IF in < DatatypeLimits.MIN_VALUE_OF_LREAL_WHICH_CAN_BE_HELD_IN_A_UDINT THEN
	RETURN;
END_IF

out := LREAL_TO_UDINT(in);
TryConvert_LREAL_TO_UDINT := TRUE;

END_FUNCTION

// ---- Converters/LREAL_TO_/TryConvert_LREAL_TO_ULINT.TcPOU
FUNCTION TryConvert_LREAL_TO_ULINT : BOOL
VAR_INPUT
	in : LREAL;
	out : REFERENCE TO ULINT;
END_VAR

IF in > DatatypeLimits.MAX_VALUE_OF_LREAL_WHICH_CAN_BE_HELD_IN_A_ULINT THEN
	RETURN;
END_IF

IF in < DatatypeLimits.MIN_VALUE_OF_LREAL_WHICH_CAN_BE_HELD_IN_A_ULINT THEN
	RETURN;
END_IF

out := LREAL_TO_ULINT(in);
TryConvert_LREAL_TO_ULINT := TRUE;

END_FUNCTION

// ---- Converters/LREAL_TO_/TryConvert_LREAL_TO_REAL.TcPOU
FUNCTION TryConvert_LREAL_TO_REAL : BOOL
VAR_INPUT
	in : LREAL;
	out : REFERENCE TO REAL;
END_VAR

IF in > DatatypeLimits.MAX_VALUE_OF_LREAL_WHICH_CAN_BE_HELD_IN_A_REAL THEN
	RETURN;
END_IF

IF in < DatatypeLimits.MIN_VALUE_OF_LREAL_WHICH_CAN_BE_HELD_IN_A_REAL THEN
	RETURN;
END_IF

out := LREAL_TO_REAL(in);
TryConvert_LREAL_TO_REAL := TRUE;

END_FUNCTION

// ---- Converters/LREAL_TO_/TryConvert_LREAL_TO_LREAL.TcPOU
FUNCTION TryConvert_LREAL_TO_LREAL : BOOL
VAR_INPUT
	in : LREAL;
	out : REFERENCE TO LREAL;
END_VAR

out := in;
TryConvert_LREAL_TO_LREAL := TRUE;

END_FUNCTION

// ---- Converters/LREAL_TO_/TryConvert_LREAL_TO_TIME.TcPOU
FUNCTION TryConvert_LREAL_TO_TIME : BOOL
VAR_INPUT
	in : LREAL;
	out : REFERENCE TO TIME;
END_VAR

IF in > DatatypeLimits.MAX_VALUE_OF_LREAL_WHICH_CAN_BE_HELD_IN_A_TIME THEN
	RETURN;
END_IF

IF in < DatatypeLimits.MIN_VALUE_OF_LREAL_WHICH_CAN_BE_HELD_IN_A_TIME THEN
	RETURN;
END_IF

out := LREAL_TO_TIME(in);
TryConvert_LREAL_TO_TIME := TRUE;

END_FUNCTION

// ---- Converters/LREAL_TO_/TryConvert_LREAL_TO_TOD.TcPOU
FUNCTION TryConvert_LREAL_TO_TOD : BOOL
VAR_INPUT
	in : LREAL;
	out : REFERENCE TO TOD;
END_VAR

IF in > DatatypeLimits.MAX_VALUE_OF_LREAL_WHICH_CAN_BE_HELD_IN_A_TOD THEN
	RETURN;
END_IF

IF in < DatatypeLimits.MIN_VALUE_OF_LREAL_WHICH_CAN_BE_HELD_IN_A_TOD THEN
	RETURN;
END_IF

out := LREAL_TO_TOD(in);
TryConvert_LREAL_TO_TOD := TRUE;

END_FUNCTION

// ---- Converters/LREAL_TO_/TryConvert_LREAL_TO_DT.TcPOU
FUNCTION TryConvert_LREAL_TO_DT : BOOL
VAR_INPUT
	in : LREAL;
	out : REFERENCE TO DT;
END_VAR

IF in > DatatypeLimits.MAX_VALUE_OF_LREAL_WHICH_CAN_BE_HELD_IN_A_DT THEN
	RETURN;
END_IF

IF in < DatatypeLimits.MIN_VALUE_OF_LREAL_WHICH_CAN_BE_HELD_IN_A_DT THEN
	RETURN;
END_IF

out := LREAL_TO_DT(in);
TryConvert_LREAL_TO_DT := TRUE;

END_FUNCTION

// ---- Converters/LREAL_TO_/TryConvert_LREAL_TO_STRING.TcPOU
FUNCTION TryConvert_LREAL_TO_STRING : BOOL
VAR_INPUT
	in : LREAL;
	out : REFERENCE TO STRING;
END_VAR

IF in > DatatypeLimits.MAX_VALUE_OF_LREAL_WHICH_CAN_BE_HELD_IN_A_STRING THEN
	RETURN;
END_IF

IF in < DatatypeLimits.MIN_VALUE_OF_LREAL_WHICH_CAN_BE_HELD_IN_A_STRING THEN
	RETURN;
END_IF

out := LREAL_TO_STRING(in);
TryConvert_LREAL_TO_STRING := TRUE;

END_FUNCTION

// ---- Converters/LWORD_TO_/TryConvert_LWORD_TO_BOOL.TcPOU
FUNCTION TryConvert_LWORD_TO_BOOL : BOOL
VAR_INPUT
	in : LWORD;
	out : REFERENCE TO BOOL;
END_VAR

out := LWORD_TO_BOOL(in);
TryConvert_LWORD_TO_BOOL := TRUE;

END_FUNCTION

// ---- Converters/LWORD_TO_/TryConvert_LWORD_TO_BYTE.TcPOU
FUNCTION TryConvert_LWORD_TO_BYTE : BOOL
VAR_INPUT
	in : LWORD;
	out : REFERENCE TO BYTE;
END_VAR

IF in > DatatypeLimits.MAX_VALUE_OF_LWORD_WHICH_CAN_BE_HELD_IN_A_BYTE THEN
	RETURN;
END_IF

out := LWORD_TO_BYTE(in);
TryConvert_LWORD_TO_BYTE := TRUE;

END_FUNCTION

// ---- Converters/LWORD_TO_/TryConvert_LWORD_TO_DATE.TcPOU
FUNCTION TryConvert_LWORD_TO_DATE : BOOL
VAR_INPUT
	in : LWORD;
	out : REFERENCE TO DATE;
END_VAR

IF in > DatatypeLimits.MAX_VALUE_OF_LWORD_WHICH_CAN_BE_HELD_IN_A_DATE THEN
	RETURN;
END_IF

out := LWORD_TO_DATE(in);
TryConvert_LWORD_TO_DATE := TRUE;

END_FUNCTION

// ---- Converters/LWORD_TO_/TryConvert_LWORD_TO_Destination.TcPOU
FUNCTION TryConvert_LWORD_TO_Destination : BOOL
VAR_INPUT
	in : LWORD;
	out : ANY;
END_VAR
VAR
	convertResult : BOOL := FALSE;
	convertAddress : PVOID;
	_BOOL : BOOL;
	_BYTE : BYTE;
	_WORD : WORD;
	_DWORD : DWORD;
	_LWORD : LWORD;
	_SINT : SINT;
	_INT : INT;
	_DINT : DINT;
	_LINT : LINT;
	_USINT : USINT;
	_UINT : UINT;
	_UDINT : UDINT;
	_ULINT : ULINT;
	_REAL : REAL;
	_LREAL : LREAL;
	_TIME : TIME;
	_TOD : TOD;
	_DATE : DATE;
	_DT : DT;
	_STRING : STRING;
END_VAR

CASE out.TypeClass OF
	__SYSTEM.TYPE_CLASS.TYPE_BOOL:
	
	convertResult := TryConvert_LWORD_TO_BOOL(in, _BOOL);
	IF convertResult THEN
		convertAddress := ADR(_BOOL);
	END_IF
	
	__SYSTEM.TYPE_CLASS.TYPE_BYTE:
	
	convertResult := TryConvert_LWORD_TO_BYTE(in, _BYTE);
	IF convertResult THEN
		convertAddress := ADR(_BYTE);
	END_IF
	
	__SYSTEM.TYPE_CLASS.TYPE_WORD:
	
	convertResult := TryConvert_LWORD_TO_WORD(in, _WORD);
	IF convertResult THEN
		convertAddress := ADR(_WORD);
	END_IF
	
	__SYSTEM.TYPE_CLASS.TYPE_DWORD:
	
	convertResult := TryConvert_LWORD_TO_DWORD(in, _DWORD);
	IF convertResult THEN
		convertAddress := ADR(_DWORD);
	END_IF
	
	__SYSTEM.TYPE_CLASS.TYPE_LWORD:
	
	convertResult := TryConvert_LWORD_TO_LWORD(in, _LWORD);
	IF convertResult THEN
		convertAddress := ADR(_LWORD);
	END_IF
	
	__SYSTEM.TYPE_CLASS.TYPE_SINT:
	
	convertResult := TryConvert_LWORD_TO_SINT(in, _SINT);
	IF convertResult THEN
		convertAddress := ADR(_SINT);
	END_IF
	
	__SYSTEM.TYPE_CLASS.TYPE_INT:
	
	convertResult := TryConvert_LWORD_TO_INT(in, _INT);
	IF convertResult THEN
		convertAddress := ADR(_INT);
	END_IF
	
	__SYSTEM.TYPE_CLASS.TYPE_DINT:
	
	convertResult := TryConvert_LWORD_TO_DINT(in, _DINT);
	IF convertResult THEN
		convertAddress := ADR(_DINT);
	END_IF
	
	__SYSTEM.TYPE_CLASS.TYPE_LINT:
	
	convertResult := TryConvert_LWORD_TO_LINT(in, _LINT);
	IF convertResult THEN
		convertAddress := ADR(_LINT);
	END_IF
	
	__SYSTEM.TYPE_CLASS.TYPE_USINT:
	
	convertResult := TryConvert_LWORD_TO_USINT(in, _USINT);
	IF convertResult THEN
		convertAddress := ADR(_USINT);
	END_IF
	
	__SYSTEM.TYPE_CLASS.TYPE_UINT:
	
	convertResult := TryConvert_LWORD_TO_UINT(in, _UINT);
	IF convertResult THEN
		convertAddress := ADR(_UINT);
	END_IF
	
	__SYSTEM.TYPE_CLASS.TYPE_UDINT:
	
	convertResult := TryConvert_LWORD_TO_UDINT(in, _UDINT);
	IF convertResult THEN
		convertAddress := ADR(_UDINT);
	END_IF
	
	__SYSTEM.TYPE_CLASS.TYPE_ULINT:
	
	convertResult := TryConvert_LWORD_TO_ULINT(in, _ULINT);
	IF convertResult THEN
		convertAddress := ADR(_ULINT);
	END_IF
	
	__SYSTEM.TYPE_CLASS.TYPE_REAL:
	
	convertResult := TryConvert_LWORD_TO_REAL(in, _REAL);
	IF convertResult THEN
		convertAddress := ADR(_REAL);
	END_IF
	
	__SYSTEM.TYPE_CLASS.TYPE_LREAL:
	
	convertResult := TryConvert_LWORD_TO_LREAL(in, _LREAL);
	IF convertResult THEN
		convertAddress := ADR(_LREAL);
	END_IF
	
	__SYSTEM.TYPE_CLASS.TYPE_TIME:
	
	convertResult := TryConvert_LWORD_TO_TIME(in, _TIME);
	IF convertResult THEN
		convertAddress := ADR(_TIME);
	END_IF
	
	__SYSTEM.TYPE_CLASS.TYPE_TIMEOFDAY:
	
	convertResult := TryConvert_LWORD_TO_TOD(in, _TOD);
	IF convertResult THEN
		convertAddress := ADR(_TOD);
	END_IF
	
	__SYSTEM.TYPE_CLASS.TYPE_DATE:
	
	convertResult := TryConvert_LWORD_TO_DATE(in, _DATE);
	IF convertResult THEN
		convertAddress := ADR(_DATE);
	END_IF
	
	__SYSTEM.TYPE_CLASS.TYPE_DATEANDTIME:
	
	convertResult := TryConvert_LWORD_TO_DT(in, _DT);
	IF convertResult THEN
		convertAddress := ADR(_DT);
	END_IF
	
	__SYSTEM.TYPE_CLASS.TYPE_STRING:
	
	convertResult := TryConvert_LWORD_TO_STRING(in, _STRING);
	IF convertResult THEN
		convertAddress := ADR(_STRING);
	END_IF
	
END_CASE

IF convertResult THEN
	memcpy(out.pValue,convertAddress,DINT_TO_UDINT(out.diSize));
END_IF

TryConvert_LWORD_TO_Destination := convertResult;

END_FUNCTION

// ---- Converters/LWORD_TO_/TryConvert_LWORD_TO_WORD.TcPOU
FUNCTION TryConvert_LWORD_TO_WORD : BOOL
VAR_INPUT
	in : LWORD;
	out : REFERENCE TO WORD;
END_VAR

IF in > DatatypeLimits.MAX_VALUE_OF_LWORD_WHICH_CAN_BE_HELD_IN_A_WORD THEN
	RETURN;
END_IF

out := LWORD_TO_WORD(in);
TryConvert_LWORD_TO_WORD := TRUE;

END_FUNCTION

// ---- Converters/LWORD_TO_/TryConvert_LWORD_TO_DWORD.TcPOU
FUNCTION TryConvert_LWORD_TO_DWORD : BOOL
VAR_INPUT
	in : LWORD;
	out : REFERENCE TO DWORD;
END_VAR

IF in > DatatypeLimits.MAX_VALUE_OF_LWORD_WHICH_CAN_BE_HELD_IN_A_DWORD THEN
	RETURN;
END_IF

out := LWORD_TO_DWORD(in);
TryConvert_LWORD_TO_DWORD := TRUE;

END_FUNCTION

// ---- Converters/LWORD_TO_/TryConvert_LWORD_TO_LWORD.TcPOU
FUNCTION TryConvert_LWORD_TO_LWORD : BOOL
VAR_INPUT
	in : LWORD;
	out : REFERENCE TO LWORD;
END_VAR

out := in;
TryConvert_LWORD_TO_LWORD := TRUE;

END_FUNCTION

// ---- Converters/LWORD_TO_/TryConvert_LWORD_TO_SINT.TcPOU
FUNCTION TryConvert_LWORD_TO_SINT : BOOL
VAR_INPUT
	in : LWORD;
	out : REFERENCE TO SINT;
END_VAR

IF in > DatatypeLimits.MAX_VALUE_OF_LWORD_WHICH_CAN_BE_HELD_IN_A_SINT THEN
	RETURN;
END_IF

out := LWORD_TO_SINT(in);
TryConvert_LWORD_TO_SINT := TRUE;

END_FUNCTION

// ---- Converters/LWORD_TO_/TryConvert_LWORD_TO_INT.TcPOU
FUNCTION TryConvert_LWORD_TO_INT : BOOL
VAR_INPUT
	in : LWORD;
	out : REFERENCE TO INT;
END_VAR

IF in > DatatypeLimits.MAX_VALUE_OF_LWORD_WHICH_CAN_BE_HELD_IN_A_INT THEN
	RETURN;
END_IF

out := LWORD_TO_INT(in);
TryConvert_LWORD_TO_INT := TRUE;

END_FUNCTION

// ---- Converters/LWORD_TO_/TryConvert_LWORD_TO_DINT.TcPOU
FUNCTION TryConvert_LWORD_TO_DINT : BOOL
VAR_INPUT
	in : LWORD;
	out : REFERENCE TO DINT;
END_VAR

IF in > DatatypeLimits.MAX_VALUE_OF_LWORD_WHICH_CAN_BE_HELD_IN_A_DINT THEN
	RETURN;
END_IF

out := LWORD_TO_DINT(in);
TryConvert_LWORD_TO_DINT := TRUE;

END_FUNCTION

// ---- Converters/LWORD_TO_/TryConvert_LWORD_TO_LINT.TcPOU
FUNCTION TryConvert_LWORD_TO_LINT : BOOL
VAR_INPUT
	in : LWORD;
	out : REFERENCE TO LINT;
END_VAR

IF in > DatatypeLimits.MAX_VALUE_OF_LWORD_WHICH_CAN_BE_HELD_IN_A_LINT THEN
	RETURN;
END_IF

out := LWORD_TO_LINT(in);
TryConvert_LWORD_TO_LINT := TRUE;

END_FUNCTION

// ---- Converters/LWORD_TO_/TryConvert_LWORD_TO_USINT.TcPOU
FUNCTION TryConvert_LWORD_TO_USINT : BOOL
VAR_INPUT
	in : LWORD;
	out : REFERENCE TO USINT;
END_VAR

IF in > DatatypeLimits.MAX_VALUE_OF_LWORD_WHICH_CAN_BE_HELD_IN_A_USINT THEN
	RETURN;
END_IF

out := LWORD_TO_USINT(in);
TryConvert_LWORD_TO_USINT := TRUE;

END_FUNCTION

// ---- Converters/LWORD_TO_/TryConvert_LWORD_TO_UINT.TcPOU
FUNCTION TryConvert_LWORD_TO_UINT : BOOL
VAR_INPUT
	in : LWORD;
	out : REFERENCE TO UINT;
END_VAR

IF in > DatatypeLimits.MAX_VALUE_OF_LWORD_WHICH_CAN_BE_HELD_IN_A_UINT THEN
	RETURN;
END_IF

out := LWORD_TO_UINT(in);
TryConvert_LWORD_TO_UINT := TRUE;

END_FUNCTION

// ---- Converters/LWORD_TO_/TryConvert_LWORD_TO_UDINT.TcPOU
FUNCTION TryConvert_LWORD_TO_UDINT : BOOL
VAR_INPUT
	in : LWORD;
	out : REFERENCE TO UDINT;
END_VAR

IF in > DatatypeLimits.MAX_VALUE_OF_LWORD_WHICH_CAN_BE_HELD_IN_A_UDINT THEN
	RETURN;
END_IF

out := LWORD_TO_UDINT(in);
TryConvert_LWORD_TO_UDINT := TRUE;

END_FUNCTION

// ---- Converters/LWORD_TO_/TryConvert_LWORD_TO_ULINT.TcPOU
FUNCTION TryConvert_LWORD_TO_ULINT : BOOL
VAR_INPUT
	in : LWORD;
	out : REFERENCE TO ULINT;
END_VAR

out := LWORD_TO_ULINT(in);
TryConvert_LWORD_TO_ULINT := TRUE;

END_FUNCTION

// ---- Converters/LWORD_TO_/TryConvert_LWORD_TO_REAL.TcPOU
FUNCTION TryConvert_LWORD_TO_REAL : BOOL
VAR_INPUT
	in : LWORD;
	out : REFERENCE TO REAL;
END_VAR

out := LWORD_TO_REAL(in);
TryConvert_LWORD_TO_REAL := TRUE;

END_FUNCTION

// ---- Converters/LWORD_TO_/TryConvert_LWORD_TO_LREAL.TcPOU
FUNCTION TryConvert_LWORD_TO_LREAL : BOOL
VAR_INPUT
	in : LWORD;
	out : REFERENCE TO LREAL;
END_VAR

out := LWORD_TO_LREAL(in);
TryConvert_LWORD_TO_LREAL := TRUE;

END_FUNCTION

// ---- Converters/LWORD_TO_/TryConvert_LWORD_TO_TIME.TcPOU
FUNCTION TryConvert_LWORD_TO_TIME : BOOL
VAR_INPUT
	in : LWORD;
	out : REFERENCE TO TIME;
END_VAR

IF in > DatatypeLimits.MAX_VALUE_OF_LWORD_WHICH_CAN_BE_HELD_IN_A_TIME THEN
	RETURN;
END_IF

out := LWORD_TO_TIME(in);
TryConvert_LWORD_TO_TIME := TRUE;

END_FUNCTION

// ---- Converters/LWORD_TO_/TryConvert_LWORD_TO_TOD.TcPOU
FUNCTION TryConvert_LWORD_TO_TOD : BOOL
VAR_INPUT
	in : LWORD;
	out : REFERENCE TO TOD;
END_VAR

IF in > DatatypeLimits.MAX_VALUE_OF_LWORD_WHICH_CAN_BE_HELD_IN_A_TOD THEN
	RETURN;
END_IF

out := LWORD_TO_TOD(in);
TryConvert_LWORD_TO_TOD := TRUE;

END_FUNCTION

// ---- Converters/LWORD_TO_/TryConvert_LWORD_TO_DT.TcPOU
FUNCTION TryConvert_LWORD_TO_DT : BOOL
VAR_INPUT
	in : LWORD;
	out : REFERENCE TO DT;
END_VAR

IF in > DatatypeLimits.MAX_VALUE_OF_LWORD_WHICH_CAN_BE_HELD_IN_A_DT THEN
	RETURN;
END_IF

out := LWORD_TO_DT(in);
TryConvert_LWORD_TO_DT := TRUE;

END_FUNCTION

// ---- Converters/LWORD_TO_/TryConvert_LWORD_TO_STRING.TcPOU
FUNCTION TryConvert_LWORD_TO_STRING : BOOL
VAR_INPUT
	in : LWORD;
	out : REFERENCE TO STRING;
END_VAR

out := LWORD_TO_STRING(in);
TryConvert_LWORD_TO_STRING := TRUE;

END_FUNCTION

// ---- Converters/REAL_TO_/TryConvert_REAL_TO_BOOL.TcPOU
FUNCTION TryConvert_REAL_TO_BOOL : BOOL
VAR_INPUT
	in : REAL;
	out : REFERENCE TO BOOL;
END_VAR

out := REAL_TO_BOOL(in);
TryConvert_REAL_TO_BOOL := TRUE;

END_FUNCTION

// ---- Converters/REAL_TO_/TryConvert_REAL_TO_BYTE.TcPOU
FUNCTION TryConvert_REAL_TO_BYTE : BOOL
VAR_INPUT
	in : REAL;
	out : REFERENCE TO BYTE;
END_VAR

IF in > DatatypeLimits.MAX_VALUE_OF_REAL_WHICH_CAN_BE_HELD_IN_A_BYTE THEN
	RETURN;
END_IF

IF in < DatatypeLimits.MIN_VALUE_OF_REAL_WHICH_CAN_BE_HELD_IN_A_BYTE THEN
	RETURN;
END_IF

out := REAL_TO_BYTE(in);
TryConvert_REAL_TO_BYTE := TRUE;

END_FUNCTION

// ---- Converters/REAL_TO_/TryConvert_REAL_TO_DATE.TcPOU
FUNCTION TryConvert_REAL_TO_DATE : BOOL
VAR_INPUT
	in : REAL;
	out : REFERENCE TO DATE;
END_VAR

IF in > DatatypeLimits.MAX_VALUE_OF_REAL_WHICH_CAN_BE_HELD_IN_A_DATE THEN
	RETURN;
END_IF

IF in < DatatypeLimits.MIN_VALUE_OF_REAL_WHICH_CAN_BE_HELD_IN_A_DATE THEN
	RETURN;
END_IF

out := REAL_TO_DATE(in);
TryConvert_REAL_TO_DATE := TRUE;

END_FUNCTION

// ---- Converters/REAL_TO_/TryConvert_REAL_TO_Destination.TcPOU
FUNCTION TryConvert_REAL_TO_Destination : BOOL
VAR_INPUT
	in : REAL;
	out : ANY;
END_VAR
VAR
	convertResult : BOOL := FALSE;
	convertAddress : PVOID;
	_BOOL : BOOL;
	_BYTE : BYTE;
	_WORD : WORD;
	_DWORD : DWORD;
	_LWORD : LWORD;
	_SINT : SINT;
	_INT : INT;
	_DINT : DINT;
	_LINT : LINT;
	_USINT : USINT;
	_UINT : UINT;
	_UDINT : UDINT;
	_ULINT : ULINT;
	_REAL : REAL;
	_LREAL : LREAL;
	_TIME : TIME;
	_TOD : TOD;
	_DATE : DATE;
	_DT : DT;
	_STRING : STRING;
END_VAR

CASE out.TypeClass OF
	__SYSTEM.TYPE_CLASS.TYPE_BOOL:
	
	convertResult := TryConvert_REAL_TO_BOOL(in, _BOOL);
	IF convertResult THEN
		convertAddress := ADR(_BOOL);
	END_IF
	
	__SYSTEM.TYPE_CLASS.TYPE_BYTE:
	
	convertResult := TryConvert_REAL_TO_BYTE(in, _BYTE);
	IF convertResult THEN
		convertAddress := ADR(_BYTE);
	END_IF
	
	__SYSTEM.TYPE_CLASS.TYPE_WORD:
	
	convertResult := TryConvert_REAL_TO_WORD(in, _WORD);
	IF convertResult THEN
		convertAddress := ADR(_WORD);
	END_IF
	
	__SYSTEM.TYPE_CLASS.TYPE_DWORD:
	
	convertResult := TryConvert_REAL_TO_DWORD(in, _DWORD);
	IF convertResult THEN
		convertAddress := ADR(_DWORD);
	END_IF
	
	__SYSTEM.TYPE_CLASS.TYPE_LWORD:
	
	convertResult := TryConvert_REAL_TO_LWORD(in, _LWORD);
	IF convertResult THEN
		convertAddress := ADR(_LWORD);
	END_IF
	
	__SYSTEM.TYPE_CLASS.TYPE_SINT:
	
	convertResult := TryConvert_REAL_TO_SINT(in, _SINT);
	IF convertResult THEN
		convertAddress := ADR(_SINT);
	END_IF
	
	__SYSTEM.TYPE_CLASS.TYPE_INT:
	
	convertResult := TryConvert_REAL_TO_INT(in, _INT);
	IF convertResult THEN
		convertAddress := ADR(_INT);
	END_IF
	
	__SYSTEM.TYPE_CLASS.TYPE_DINT:
	
	convertResult := TryConvert_REAL_TO_DINT(in, _DINT);
	IF convertResult THEN
		convertAddress := ADR(_DINT);
	END_IF
	
	__SYSTEM.TYPE_CLASS.TYPE_LINT:
	
	convertResult := TryConvert_REAL_TO_LINT(in, _LINT);
	IF convertResult THEN
		convertAddress := ADR(_LINT);
	END_IF
	
	__SYSTEM.TYPE_CLASS.TYPE_USINT:
	
	convertResult := TryConvert_REAL_TO_USINT(in, _USINT);
	IF convertResult THEN
		convertAddress := ADR(_USINT);
	END_IF
	
	__SYSTEM.TYPE_CLASS.TYPE_UINT:
	
	convertResult := TryConvert_REAL_TO_UINT(in, _UINT);
	IF convertResult THEN
		convertAddress := ADR(_UINT);
	END_IF
	
	__SYSTEM.TYPE_CLASS.TYPE_UDINT:
	
	convertResult := TryConvert_REAL_TO_UDINT(in, _UDINT);
	IF convertResult THEN
		convertAddress := ADR(_UDINT);
	END_IF
	
	__SYSTEM.TYPE_CLASS.TYPE_ULINT:
	
	convertResult := TryConvert_REAL_TO_ULINT(in, _ULINT);
	IF convertResult THEN
		convertAddress := ADR(_ULINT);
	END_IF
	
	__SYSTEM.TYPE_CLASS.TYPE_REAL:
	
	convertResult := TryConvert_REAL_TO_REAL(in, _REAL);
	IF convertResult THEN
		convertAddress := ADR(_REAL);
	END_IF
	
	__SYSTEM.TYPE_CLASS.TYPE_LREAL:
	
	convertResult := TryConvert_REAL_TO_LREAL(in, _LREAL);
	IF convertResult THEN
		convertAddress := ADR(_LREAL);
	END_IF
	
	__SYSTEM.TYPE_CLASS.TYPE_TIME:
	
	convertResult := TryConvert_REAL_TO_TIME(in, _TIME);
	IF convertResult THEN
		convertAddress := ADR(_TIME);
	END_IF
	
	__SYSTEM.TYPE_CLASS.TYPE_TIMEOFDAY:
	
	convertResult := TryConvert_REAL_TO_TOD(in, _TOD);
	IF convertResult THEN
		convertAddress := ADR(_TOD);
	END_IF
	
	__SYSTEM.TYPE_CLASS.TYPE_DATE:
	
	convertResult := TryConvert_REAL_TO_DATE(in, _DATE);
	IF convertResult THEN
		convertAddress := ADR(_DATE);
	END_IF
	
	__SYSTEM.TYPE_CLASS.TYPE_DATEANDTIME:
	
	convertResult := TryConvert_REAL_TO_DT(in, _DT);
	IF convertResult THEN
		convertAddress := ADR(_DT);
	END_IF
	
	__SYSTEM.TYPE_CLASS.TYPE_STRING:
	
	convertResult := TryConvert_REAL_TO_STRING(in, _STRING);
	IF convertResult THEN
		convertAddress := ADR(_STRING);
	END_IF
	
END_CASE

IF convertResult THEN
	memcpy(out.pValue,convertAddress,DINT_TO_UDINT(out.diSize));
END_IF

TryConvert_REAL_TO_Destination := convertResult;

END_FUNCTION

// ---- Converters/REAL_TO_/TryConvert_REAL_TO_WORD.TcPOU
FUNCTION TryConvert_REAL_TO_WORD : BOOL
VAR_INPUT
	in : REAL;
	out : REFERENCE TO WORD;
END_VAR

IF in > DatatypeLimits.MAX_VALUE_OF_REAL_WHICH_CAN_BE_HELD_IN_A_WORD THEN
	RETURN;
END_IF

IF in < DatatypeLimits.MIN_VALUE_OF_REAL_WHICH_CAN_BE_HELD_IN_A_WORD THEN
	RETURN;
END_IF

out := REAL_TO_WORD(in);
TryConvert_REAL_TO_WORD := TRUE;

END_FUNCTION

// ---- Converters/REAL_TO_/TryConvert_REAL_TO_DWORD.TcPOU
FUNCTION TryConvert_REAL_TO_DWORD : BOOL
VAR_INPUT
	in : REAL;
	out : REFERENCE TO DWORD;
END_VAR

IF in > DatatypeLimits.MAX_VALUE_OF_REAL_WHICH_CAN_BE_HELD_IN_A_DWORD THEN
	RETURN;
END_IF

IF in < DatatypeLimits.MIN_VALUE_OF_REAL_WHICH_CAN_BE_HELD_IN_A_DWORD THEN
	RETURN;
END_IF

out := REAL_TO_DWORD(in);
TryConvert_REAL_TO_DWORD := TRUE;

END_FUNCTION

// ---- Converters/REAL_TO_/TryConvert_REAL_TO_LWORD.TcPOU
FUNCTION TryConvert_REAL_TO_LWORD : BOOL
VAR_INPUT
	in : REAL;
	out : REFERENCE TO LWORD;
END_VAR

IF in > DatatypeLimits.MAX_VALUE_OF_REAL_WHICH_CAN_BE_HELD_IN_A_LWORD THEN
	RETURN;
END_IF

IF in < DatatypeLimits.MIN_VALUE_OF_REAL_WHICH_CAN_BE_HELD_IN_A_LWORD THEN
	RETURN;
END_IF

out := REAL_TO_LWORD(in);
TryConvert_REAL_TO_LWORD := TRUE;

END_FUNCTION

// ---- Converters/REAL_TO_/TryConvert_REAL_TO_SINT.TcPOU
FUNCTION TryConvert_REAL_TO_SINT : BOOL
VAR_INPUT
	in : REAL;
	out : REFERENCE TO SINT;
END_VAR

IF in > DatatypeLimits.MAX_VALUE_OF_REAL_WHICH_CAN_BE_HELD_IN_A_SINT THEN
	RETURN;
END_IF

IF in < DatatypeLimits.MIN_VALUE_OF_REAL_WHICH_CAN_BE_HELD_IN_A_SINT THEN
	RETURN;
END_IF

out := REAL_TO_SINT(in);
TryConvert_REAL_TO_SINT := TRUE;

END_FUNCTION

// ---- Converters/REAL_TO_/TryConvert_REAL_TO_INT.TcPOU
FUNCTION TryConvert_REAL_TO_INT : BOOL
VAR_INPUT
	in : REAL;
	out : REFERENCE TO INT;
END_VAR

IF in > DatatypeLimits.MAX_VALUE_OF_REAL_WHICH_CAN_BE_HELD_IN_A_INT THEN
	RETURN;
END_IF

IF in < DatatypeLimits.MIN_VALUE_OF_REAL_WHICH_CAN_BE_HELD_IN_A_INT THEN
	RETURN;
END_IF

out := REAL_TO_INT(in);
TryConvert_REAL_TO_INT := TRUE;

END_FUNCTION

// ---- Converters/REAL_TO_/TryConvert_REAL_TO_DINT.TcPOU
FUNCTION TryConvert_REAL_TO_DINT : BOOL
VAR_INPUT
	in : REAL;
	out : REFERENCE TO DINT;
END_VAR

IF in > DatatypeLimits.MAX_VALUE_OF_REAL_WHICH_CAN_BE_HELD_IN_A_DINT THEN
	RETURN;
END_IF

IF in < DatatypeLimits.MIN_VALUE_OF_REAL_WHICH_CAN_BE_HELD_IN_A_DINT THEN
	RETURN;
END_IF

out := REAL_TO_DINT(in);
TryConvert_REAL_TO_DINT := TRUE;

END_FUNCTION

// ---- Converters/REAL_TO_/TryConvert_REAL_TO_LINT.TcPOU
FUNCTION TryConvert_REAL_TO_LINT : BOOL
VAR_INPUT
	in : REAL;
	out : REFERENCE TO LINT;
END_VAR

IF in > DatatypeLimits.MAX_VALUE_OF_REAL_WHICH_CAN_BE_HELD_IN_A_LINT THEN
	RETURN;
END_IF

IF in < DatatypeLimits.MIN_VALUE_OF_REAL_WHICH_CAN_BE_HELD_IN_A_LINT THEN
	RETURN;
END_IF

out := REAL_TO_LINT(in);
TryConvert_REAL_TO_LINT := TRUE;

END_FUNCTION

// ---- Converters/REAL_TO_/TryConvert_REAL_TO_USINT.TcPOU
FUNCTION TryConvert_REAL_TO_USINT : BOOL
VAR_INPUT
	in : REAL;
	out : REFERENCE TO USINT;
END_VAR

IF in > DatatypeLimits.MAX_VALUE_OF_REAL_WHICH_CAN_BE_HELD_IN_A_USINT THEN
	RETURN;
END_IF

IF in < DatatypeLimits.MIN_VALUE_OF_REAL_WHICH_CAN_BE_HELD_IN_A_USINT THEN
	RETURN;
END_IF

out := REAL_TO_USINT(in);
TryConvert_REAL_TO_USINT := TRUE;

END_FUNCTION

// ---- Converters/REAL_TO_/TryConvert_REAL_TO_UINT.TcPOU
FUNCTION TryConvert_REAL_TO_UINT : BOOL
VAR_INPUT
	in : REAL;
	out : REFERENCE TO UINT;
END_VAR

IF in > DatatypeLimits.MAX_VALUE_OF_REAL_WHICH_CAN_BE_HELD_IN_A_UINT THEN
	RETURN;
END_IF

IF in < DatatypeLimits.MIN_VALUE_OF_REAL_WHICH_CAN_BE_HELD_IN_A_UINT THEN
	RETURN;
END_IF

out := REAL_TO_UINT(in);
TryConvert_REAL_TO_UINT := TRUE;

END_FUNCTION

// ---- Converters/REAL_TO_/TryConvert_REAL_TO_UDINT.TcPOU
FUNCTION TryConvert_REAL_TO_UDINT : BOOL
VAR_INPUT
	in : REAL;
	out : REFERENCE TO UDINT;
END_VAR

IF in > DatatypeLimits.MAX_VALUE_OF_REAL_WHICH_CAN_BE_HELD_IN_A_UDINT THEN
	RETURN;
END_IF

IF in < DatatypeLimits.MIN_VALUE_OF_REAL_WHICH_CAN_BE_HELD_IN_A_UDINT THEN
	RETURN;
END_IF

out := REAL_TO_UDINT(in);
TryConvert_REAL_TO_UDINT := TRUE;

END_FUNCTION

// ---- Converters/REAL_TO_/TryConvert_REAL_TO_ULINT.TcPOU
FUNCTION TryConvert_REAL_TO_ULINT : BOOL
VAR_INPUT
	in : REAL;
	out : REFERENCE TO ULINT;
END_VAR

IF in > DatatypeLimits.MAX_VALUE_OF_REAL_WHICH_CAN_BE_HELD_IN_A_ULINT THEN
	RETURN;
END_IF

IF in < DatatypeLimits.MIN_VALUE_OF_REAL_WHICH_CAN_BE_HELD_IN_A_ULINT THEN
	RETURN;
END_IF

out := REAL_TO_ULINT(in);
TryConvert_REAL_TO_ULINT := TRUE;

END_FUNCTION

// ---- Converters/REAL_TO_/TryConvert_REAL_TO_REAL.TcPOU
FUNCTION TryConvert_REAL_TO_REAL : BOOL
VAR_INPUT
	in : REAL;
	out : REFERENCE TO REAL;
END_VAR

out := in;
TryConvert_REAL_TO_REAL := TRUE;

END_FUNCTION

// ---- Converters/REAL_TO_/TryConvert_REAL_TO_LREAL.TcPOU
FUNCTION TryConvert_REAL_TO_LREAL : BOOL
VAR_INPUT
	in : REAL;
	out : REFERENCE TO LREAL;
END_VAR

out := REAL_TO_LREAL(in);
TryConvert_REAL_TO_LREAL := TRUE;

END_FUNCTION

// ---- Converters/REAL_TO_/TryConvert_REAL_TO_TIME.TcPOU
FUNCTION TryConvert_REAL_TO_TIME : BOOL
VAR_INPUT
	in : REAL;
	out : REFERENCE TO TIME;
END_VAR

IF in > DatatypeLimits.MAX_VALUE_OF_REAL_WHICH_CAN_BE_HELD_IN_A_TIME THEN
	RETURN;
END_IF

IF in < DatatypeLimits.MIN_VALUE_OF_REAL_WHICH_CAN_BE_HELD_IN_A_TIME THEN
	RETURN;
END_IF

out := REAL_TO_TIME(in);
TryConvert_REAL_TO_TIME := TRUE;

END_FUNCTION

// ---- Converters/REAL_TO_/TryConvert_REAL_TO_TOD.TcPOU
FUNCTION TryConvert_REAL_TO_TOD : BOOL
VAR_INPUT
	in : REAL;
	out : REFERENCE TO TOD;
END_VAR

IF in > DatatypeLimits.MAX_VALUE_OF_REAL_WHICH_CAN_BE_HELD_IN_A_TOD THEN
	RETURN;
END_IF

IF in < DatatypeLimits.MIN_VALUE_OF_REAL_WHICH_CAN_BE_HELD_IN_A_TOD THEN
	RETURN;
END_IF

out := REAL_TO_TOD(in);
TryConvert_REAL_TO_TOD := TRUE;

END_FUNCTION

// ---- Converters/REAL_TO_/TryConvert_REAL_TO_DT.TcPOU
FUNCTION TryConvert_REAL_TO_DT : BOOL
VAR_INPUT
	in : REAL;
	out : REFERENCE TO DT;
END_VAR

IF in > DatatypeLimits.MAX_VALUE_OF_REAL_WHICH_CAN_BE_HELD_IN_A_DT THEN
	RETURN;
END_IF

IF in < DatatypeLimits.MIN_VALUE_OF_REAL_WHICH_CAN_BE_HELD_IN_A_DT THEN
	RETURN;
END_IF

out := REAL_TO_DT(in);
TryConvert_REAL_TO_DT := TRUE;

END_FUNCTION

// ---- Converters/REAL_TO_/TryConvert_REAL_TO_STRING.TcPOU
FUNCTION TryConvert_REAL_TO_STRING : BOOL
VAR_INPUT
	in : REAL;
	out : REFERENCE TO STRING;
END_VAR

out := REAL_TO_STRING(in);
TryConvert_REAL_TO_STRING := TRUE;

END_FUNCTION

// ---- Converters/SINT_TO_/TryConvert_SINT_TO_BOOL.TcPOU
FUNCTION TryConvert_SINT_TO_BOOL : BOOL
VAR_INPUT
	in : SINT;
	out : REFERENCE TO BOOL;
END_VAR

out := SINT_TO_BOOL(in);
TryConvert_SINT_TO_BOOL := TRUE;

END_FUNCTION

// ---- Converters/SINT_TO_/TryConvert_SINT_TO_BYTE.TcPOU
FUNCTION TryConvert_SINT_TO_BYTE : BOOL
VAR_INPUT
	in : SINT;
	out : REFERENCE TO BYTE;
END_VAR

IF in < DatatypeLimits.MIN_VALUE_OF_SINT_WHICH_CAN_BE_HELD_IN_A_BYTE THEN
	RETURN;
END_IF

out := SINT_TO_BYTE(in);
TryConvert_SINT_TO_BYTE := TRUE;

END_FUNCTION

// ---- Converters/SINT_TO_/TryConvert_SINT_TO_DATE.TcPOU
FUNCTION TryConvert_SINT_TO_DATE : BOOL
VAR_INPUT
	in : SINT;
	out : REFERENCE TO DATE;
END_VAR

IF in < DatatypeLimits.MIN_VALUE_OF_SINT_WHICH_CAN_BE_HELD_IN_A_DATE THEN
	RETURN;
END_IF

out := SINT_TO_DATE(in);
TryConvert_SINT_TO_DATE := TRUE;

END_FUNCTION

// ---- Converters/SINT_TO_/TryConvert_SINT_TO_Destination.TcPOU
FUNCTION TryConvert_SINT_TO_Destination : BOOL
VAR_INPUT
	in : SINT;
	out : ANY;
END_VAR
VAR
	convertResult : BOOL := FALSE;
	convertAddress : PVOID;
	_BOOL : BOOL;
	_BYTE : BYTE;
	_WORD : WORD;
	_DWORD : DWORD;
	_LWORD : LWORD;
	_SINT : SINT;
	_INT : INT;
	_DINT : DINT;
	_LINT : LINT;
	_USINT : USINT;
	_UINT : UINT;
	_UDINT : UDINT;
	_ULINT : ULINT;
	_REAL : REAL;
	_LREAL : LREAL;
	_TIME : TIME;
	_TOD : TOD;
	_DATE : DATE;
	_DT : DT;
	_STRING : STRING;
END_VAR

CASE out.TypeClass OF
	__SYSTEM.TYPE_CLASS.TYPE_BOOL:
	
	convertResult := TryConvert_SINT_TO_BOOL(in, _BOOL);
	IF convertResult THEN
		convertAddress := ADR(_BOOL);
	END_IF
	
	__SYSTEM.TYPE_CLASS.TYPE_BYTE:
	
	convertResult := TryConvert_SINT_TO_BYTE(in, _BYTE);
	IF convertResult THEN
		convertAddress := ADR(_BYTE);
	END_IF
	
	__SYSTEM.TYPE_CLASS.TYPE_WORD:
	
	convertResult := TryConvert_SINT_TO_WORD(in, _WORD);
	IF convertResult THEN
		convertAddress := ADR(_WORD);
	END_IF
	
	__SYSTEM.TYPE_CLASS.TYPE_DWORD:
	
	convertResult := TryConvert_SINT_TO_DWORD(in, _DWORD);
	IF convertResult THEN
		convertAddress := ADR(_DWORD);
	END_IF
	
	__SYSTEM.TYPE_CLASS.TYPE_LWORD:
	
	convertResult := TryConvert_SINT_TO_LWORD(in, _LWORD);
	IF convertResult THEN
		convertAddress := ADR(_LWORD);
	END_IF
	
	__SYSTEM.TYPE_CLASS.TYPE_SINT:
	
	convertResult := TryConvert_SINT_TO_SINT(in, _SINT);
	IF convertResult THEN
		convertAddress := ADR(_SINT);
	END_IF
	
	__SYSTEM.TYPE_CLASS.TYPE_INT:
	
	convertResult := TryConvert_SINT_TO_INT(in, _INT);
	IF convertResult THEN
		convertAddress := ADR(_INT);
	END_IF
	
	__SYSTEM.TYPE_CLASS.TYPE_DINT:
	
	convertResult := TryConvert_SINT_TO_DINT(in, _DINT);
	IF convertResult THEN
		convertAddress := ADR(_DINT);
	END_IF
	
	__SYSTEM.TYPE_CLASS.TYPE_LINT:
	
	convertResult := TryConvert_SINT_TO_LINT(in, _LINT);
	IF convertResult THEN
		convertAddress := ADR(_LINT);
	END_IF
	
	__SYSTEM.TYPE_CLASS.TYPE_USINT:
	
	convertResult := TryConvert_SINT_TO_USINT(in, _USINT);
	IF convertResult THEN
		convertAddress := ADR(_USINT);
	END_IF
	
	__SYSTEM.TYPE_CLASS.TYPE_UINT:
	
	convertResult := TryConvert_SINT_TO_UINT(in, _UINT);
	IF convertResult THEN
		convertAddress := ADR(_UINT);
	END_IF
	
	__SYSTEM.TYPE_CLASS.TYPE_UDINT:
	
	convertResult := TryConvert_SINT_TO_UDINT(in, _UDINT);
	IF convertResult THEN
		convertAddress := ADR(_UDINT);
	END_IF
	
	__SYSTEM.TYPE_CLASS.TYPE_ULINT:
	
	convertResult := TryConvert_SINT_TO_ULINT(in, _ULINT);
	IF convertResult THEN
		convertAddress := ADR(_ULINT);
	END_IF
	
	__SYSTEM.TYPE_CLASS.TYPE_REAL:
	
	convertResult := TryConvert_SINT_TO_REAL(in, _REAL);
	IF convertResult THEN
		convertAddress := ADR(_REAL);
	END_IF
	
	__SYSTEM.TYPE_CLASS.TYPE_LREAL:
	
	convertResult := TryConvert_SINT_TO_LREAL(in, _LREAL);
	IF convertResult THEN
		convertAddress := ADR(_LREAL);
	END_IF
	
	__SYSTEM.TYPE_CLASS.TYPE_TIME:
	
	convertResult := TryConvert_SINT_TO_TIME(in, _TIME);
	IF convertResult THEN
		convertAddress := ADR(_TIME);
	END_IF
	
	__SYSTEM.TYPE_CLASS.TYPE_TIMEOFDAY:
	
	convertResult := TryConvert_SINT_TO_TOD(in, _TOD);
	IF convertResult THEN
		convertAddress := ADR(_TOD);
	END_IF
	
	__SYSTEM.TYPE_CLASS.TYPE_DATE:
	
	convertResult := TryConvert_SINT_TO_DATE(in, _DATE);
	IF convertResult THEN
		convertAddress := ADR(_DATE);
	END_IF
	
	__SYSTEM.TYPE_CLASS.TYPE_DATEANDTIME:
	
	convertResult := TryConvert_SINT_TO_DT(in, _DT);
	IF convertResult THEN
		convertAddress := ADR(_DT);
	END_IF
	
	__SYSTEM.TYPE_CLASS.TYPE_STRING:
	
	convertResult := TryConvert_SINT_TO_STRING(in, _STRING);
	IF convertResult THEN
		convertAddress := ADR(_STRING);
	END_IF
	
END_CASE

IF convertResult THEN
	memcpy(out.pValue,convertAddress,DINT_TO_UDINT(out.diSize));
END_IF

TryConvert_SINT_TO_Destination := convertResult;

END_FUNCTION

// ---- Converters/SINT_TO_/TryConvert_SINT_TO_WORD.TcPOU
FUNCTION TryConvert_SINT_TO_WORD : BOOL
VAR_INPUT
	in : SINT;
	out : REFERENCE TO WORD;
END_VAR

IF in < DatatypeLimits.MIN_VALUE_OF_SINT_WHICH_CAN_BE_HELD_IN_A_WORD THEN
	RETURN;
END_IF

out := SINT_TO_WORD(in);
TryConvert_SINT_TO_WORD := TRUE;

END_FUNCTION

// ---- Converters/SINT_TO_/TryConvert_SINT_TO_DWORD.TcPOU
FUNCTION TryConvert_SINT_TO_DWORD : BOOL
VAR_INPUT
	in : SINT;
	out : REFERENCE TO DWORD;
END_VAR

IF in < DatatypeLimits.MIN_VALUE_OF_SINT_WHICH_CAN_BE_HELD_IN_A_DWORD THEN
	RETURN;
END_IF

out := SINT_TO_DWORD(in);
TryConvert_SINT_TO_DWORD := TRUE;

END_FUNCTION

// ---- Converters/SINT_TO_/TryConvert_SINT_TO_LWORD.TcPOU
FUNCTION TryConvert_SINT_TO_LWORD : BOOL
VAR_INPUT
	in : SINT;
	out : REFERENCE TO LWORD;
END_VAR

IF in < DatatypeLimits.MIN_VALUE_OF_SINT_WHICH_CAN_BE_HELD_IN_A_LWORD THEN
	RETURN;
END_IF

out := SINT_TO_LWORD(in);
TryConvert_SINT_TO_LWORD := TRUE;

END_FUNCTION

// ---- Converters/SINT_TO_/TryConvert_SINT_TO_SINT.TcPOU
FUNCTION TryConvert_SINT_TO_SINT : BOOL
VAR_INPUT
	in : SINT;
	out : REFERENCE TO SINT;
END_VAR

out := in;
TryConvert_SINT_TO_SINT := TRUE;

END_FUNCTION

// ---- Converters/SINT_TO_/TryConvert_SINT_TO_INT.TcPOU
FUNCTION TryConvert_SINT_TO_INT : BOOL
VAR_INPUT
	in : SINT;
	out : REFERENCE TO INT;
END_VAR

out := SINT_TO_INT(in);
TryConvert_SINT_TO_INT := TRUE;

END_FUNCTION

// ---- Converters/SINT_TO_/TryConvert_SINT_TO_DINT.TcPOU
FUNCTION TryConvert_SINT_TO_DINT : BOOL
VAR_INPUT
	in : SINT;
	out : REFERENCE TO DINT;
END_VAR

out := SINT_TO_DINT(in);
TryConvert_SINT_TO_DINT := TRUE;

END_FUNCTION

// ---- Converters/SINT_TO_/TryConvert_SINT_TO_LINT.TcPOU
FUNCTION TryConvert_SINT_TO_LINT : BOOL
VAR_INPUT
	in : SINT;
	out : REFERENCE TO LINT;
END_VAR

out := SINT_TO_LINT(in);
TryConvert_SINT_TO_LINT := TRUE;

END_FUNCTION

// ---- Converters/SINT_TO_/TryConvert_SINT_TO_USINT.TcPOU
FUNCTION TryConvert_SINT_TO_USINT : BOOL
VAR_INPUT
	in : SINT;
	out : REFERENCE TO USINT;
END_VAR

IF in < DatatypeLimits.MIN_VALUE_OF_SINT_WHICH_CAN_BE_HELD_IN_A_USINT THEN
	RETURN;
END_IF

out := SINT_TO_USINT(in);
TryConvert_SINT_TO_USINT := TRUE;

END_FUNCTION

// ---- Converters/SINT_TO_/TryConvert_SINT_TO_UINT.TcPOU
FUNCTION TryConvert_SINT_TO_UINT : BOOL
VAR_INPUT
	in : SINT;
	out : REFERENCE TO UINT;
END_VAR

IF in < DatatypeLimits.MIN_VALUE_OF_SINT_WHICH_CAN_BE_HELD_IN_A_UINT THEN
	RETURN;
END_IF

out := SINT_TO_UINT(in);
TryConvert_SINT_TO_UINT := TRUE;

END_FUNCTION

// ---- Converters/SINT_TO_/TryConvert_SINT_TO_UDINT.TcPOU
FUNCTION TryConvert_SINT_TO_UDINT : BOOL
VAR_INPUT
	in : SINT;
	out : REFERENCE TO UDINT;
END_VAR

IF in < DatatypeLimits.MIN_VALUE_OF_SINT_WHICH_CAN_BE_HELD_IN_A_UDINT THEN
	RETURN;
END_IF

out := SINT_TO_UDINT(in);
TryConvert_SINT_TO_UDINT := TRUE;

END_FUNCTION

// ---- Converters/SINT_TO_/TryConvert_SINT_TO_ULINT.TcPOU
FUNCTION TryConvert_SINT_TO_ULINT : BOOL
VAR_INPUT
	in : SINT;
	out : REFERENCE TO ULINT;
END_VAR

IF in < DatatypeLimits.MIN_VALUE_OF_SINT_WHICH_CAN_BE_HELD_IN_A_ULINT THEN
	RETURN;
END_IF

out := SINT_TO_ULINT(in);
TryConvert_SINT_TO_ULINT := TRUE;

END_FUNCTION

// ---- Converters/SINT_TO_/TryConvert_SINT_TO_REAL.TcPOU
FUNCTION TryConvert_SINT_TO_REAL : BOOL
VAR_INPUT
	in : SINT;
	out : REFERENCE TO REAL;
END_VAR

out := SINT_TO_REAL(in);
TryConvert_SINT_TO_REAL := TRUE;

END_FUNCTION

// ---- Converters/SINT_TO_/TryConvert_SINT_TO_LREAL.TcPOU
FUNCTION TryConvert_SINT_TO_LREAL : BOOL
VAR_INPUT
	in : SINT;
	out : REFERENCE TO LREAL;
END_VAR

out := SINT_TO_LREAL(in);
TryConvert_SINT_TO_LREAL := TRUE;

END_FUNCTION

// ---- Converters/SINT_TO_/TryConvert_SINT_TO_TIME.TcPOU
FUNCTION TryConvert_SINT_TO_TIME : BOOL
VAR_INPUT
	in : SINT;
	out : REFERENCE TO TIME;
END_VAR

IF in < DatatypeLimits.MIN_VALUE_OF_SINT_WHICH_CAN_BE_HELD_IN_A_TIME THEN
	RETURN;
END_IF

out := SINT_TO_TIME(in);
TryConvert_SINT_TO_TIME := TRUE;

END_FUNCTION

// ---- Converters/SINT_TO_/TryConvert_SINT_TO_TOD.TcPOU
FUNCTION TryConvert_SINT_TO_TOD : BOOL
VAR_INPUT
	in : SINT;
	out : REFERENCE TO TOD;
END_VAR

IF in < DatatypeLimits.MIN_VALUE_OF_SINT_WHICH_CAN_BE_HELD_IN_A_TOD THEN
	RETURN;
END_IF

out := SINT_TO_TOD(in);
TryConvert_SINT_TO_TOD := TRUE;

END_FUNCTION

// ---- Converters/SINT_TO_/TryConvert_SINT_TO_DT.TcPOU
FUNCTION TryConvert_SINT_TO_DT : BOOL
VAR_INPUT
	in : SINT;
	out : REFERENCE TO DT;
END_VAR

IF in < DatatypeLimits.MIN_VALUE_OF_SINT_WHICH_CAN_BE_HELD_IN_A_DT THEN
	RETURN;
END_IF

out := SINT_TO_DT(in);
TryConvert_SINT_TO_DT := TRUE;

END_FUNCTION

// ---- Converters/SINT_TO_/TryConvert_SINT_TO_STRING.TcPOU
FUNCTION TryConvert_SINT_TO_STRING : BOOL
VAR_INPUT
	in : SINT;
	out : REFERENCE TO STRING;
END_VAR

out := SINT_TO_STRING(in);
TryConvert_SINT_TO_STRING := TRUE;

END_FUNCTION

// ---- Converters/STRING_TO_/TryConvert_STRING_TO_BOOL.TcPOU
FUNCTION TryConvert_STRING_TO_BOOL : BOOL
VAR_INPUT
	in : STRING;
	out : REFERENCE TO BOOL;
END_VAR

out := STRING_TO_BOOL(in);
TryConvert_STRING_TO_BOOL := TRUE;

END_FUNCTION

// ---- Converters/STRING_TO_/TryConvert_STRING_TO_BYTE.TcPOU
FUNCTION TryConvert_STRING_TO_BYTE : BOOL
VAR_INPUT
	in : STRING;
	out : REFERENCE TO BYTE;
END_VAR

IF in <> BYTE_TO_STRING(STRING_TO_BYTE(in)) THEN
	RETURN;
END_IF

out := STRING_TO_BYTE(in);
TryConvert_STRING_TO_BYTE := TRUE;

END_FUNCTION

// ---- Converters/STRING_TO_/TryConvert_STRING_TO_DATE.TcPOU
FUNCTION TryConvert_STRING_TO_DATE : BOOL
VAR_INPUT
	in : STRING;
	out : REFERENCE TO DATE;
END_VAR

IF in <> DATE_TO_STRING(STRING_TO_DATE(in)) THEN
	RETURN;
END_IF

out := STRING_TO_DATE(in);
TryConvert_STRING_TO_DATE := TRUE;

END_FUNCTION

// ---- Converters/STRING_TO_/TryConvert_STRING_TO_Destination.TcPOU
FUNCTION TryConvert_STRING_TO_Destination : BOOL
VAR_INPUT
	in : STRING;
	out : ANY;
END_VAR
VAR
	convertResult : BOOL := FALSE;
	convertAddress : PVOID;
	_BOOL : BOOL;
	_BYTE : BYTE;
	_WORD : WORD;
	_DWORD : DWORD;
	_LWORD : LWORD;
	_SINT : SINT;
	_INT : INT;
	_DINT : DINT;
	_LINT : LINT;
	_USINT : USINT;
	_UINT : UINT;
	_UDINT : UDINT;
	_ULINT : ULINT;
	_REAL : REAL;
	_LREAL : LREAL;
	_TIME : TIME;
	_TOD : TOD;
	_DATE : DATE;
	_DT : DT;
	_STRING : STRING;
END_VAR

CASE out.TypeClass OF
	__SYSTEM.TYPE_CLASS.TYPE_BOOL:
	
	convertResult := TryConvert_STRING_TO_BOOL(in, _BOOL);
	IF convertResult THEN
		convertAddress := ADR(_BOOL);
	END_IF
	
	__SYSTEM.TYPE_CLASS.TYPE_BYTE:
	
	convertResult := TryConvert_STRING_TO_BYTE(in, _BYTE);
	IF convertResult THEN
		convertAddress := ADR(_BYTE);
	END_IF
	
	__SYSTEM.TYPE_CLASS.TYPE_WORD:
	
	convertResult := TryConvert_STRING_TO_WORD(in, _WORD);
	IF convertResult THEN
		convertAddress := ADR(_WORD);
	END_IF
	
	__SYSTEM.TYPE_CLASS.TYPE_DWORD:
	
	convertResult := TryConvert_STRING_TO_DWORD(in, _DWORD);
	IF convertResult THEN
		convertAddress := ADR(_DWORD);
	END_IF
	
	__SYSTEM.TYPE_CLASS.TYPE_LWORD:
	
	convertResult := TryConvert_STRING_TO_LWORD(in, _LWORD);
	IF convertResult THEN
		convertAddress := ADR(_LWORD);
	END_IF
	
	__SYSTEM.TYPE_CLASS.TYPE_SINT:
	
	convertResult := TryConvert_STRING_TO_SINT(in, _SINT);
	IF convertResult THEN
		convertAddress := ADR(_SINT);
	END_IF
	
	__SYSTEM.TYPE_CLASS.TYPE_INT:
	
	convertResult := TryConvert_STRING_TO_INT(in, _INT);
	IF convertResult THEN
		convertAddress := ADR(_INT);
	END_IF
	
	__SYSTEM.TYPE_CLASS.TYPE_DINT:
	
	convertResult := TryConvert_STRING_TO_DINT(in, _DINT);
	IF convertResult THEN
		convertAddress := ADR(_DINT);
	END_IF
	
	__SYSTEM.TYPE_CLASS.TYPE_LINT:
	
	convertResult := TryConvert_STRING_TO_LINT(in, _LINT);
	IF convertResult THEN
		convertAddress := ADR(_LINT);
	END_IF
	
	__SYSTEM.TYPE_CLASS.TYPE_USINT:
	
	convertResult := TryConvert_STRING_TO_USINT(in, _USINT);
	IF convertResult THEN
		convertAddress := ADR(_USINT);
	END_IF
	
	__SYSTEM.TYPE_CLASS.TYPE_UINT:
	
	convertResult := TryConvert_STRING_TO_UINT(in, _UINT);
	IF convertResult THEN
		convertAddress := ADR(_UINT);
	END_IF
	
	__SYSTEM.TYPE_CLASS.TYPE_UDINT:
	
	convertResult := TryConvert_STRING_TO_UDINT(in, _UDINT);
	IF convertResult THEN
		convertAddress := ADR(_UDINT);
	END_IF
	
	__SYSTEM.TYPE_CLASS.TYPE_ULINT:
	
	convertResult := TryConvert_STRING_TO_ULINT(in, _ULINT);
	IF convertResult THEN
		convertAddress := ADR(_ULINT);
	END_IF
	
	__SYSTEM.TYPE_CLASS.TYPE_REAL:
	
	convertResult := TryConvert_STRING_TO_REAL(in, _REAL);
	IF convertResult THEN
		convertAddress := ADR(_REAL);
	END_IF
	
	__SYSTEM.TYPE_CLASS.TYPE_LREAL:
	
	convertResult := TryConvert_STRING_TO_LREAL(in, _LREAL);
	IF convertResult THEN
		convertAddress := ADR(_LREAL);
	END_IF
	
	__SYSTEM.TYPE_CLASS.TYPE_TIME:
	
	convertResult := TryConvert_STRING_TO_TIME(in, _TIME);
	IF convertResult THEN
		convertAddress := ADR(_TIME);
	END_IF
	
	__SYSTEM.TYPE_CLASS.TYPE_TIMEOFDAY:
	
	convertResult := TryConvert_STRING_TO_TOD(in, _TOD);
	IF convertResult THEN
		convertAddress := ADR(_TOD);
	END_IF
	
	__SYSTEM.TYPE_CLASS.TYPE_DATE:
	
	convertResult := TryConvert_STRING_TO_DATE(in, _DATE);
	IF convertResult THEN
		convertAddress := ADR(_DATE);
	END_IF
	
	__SYSTEM.TYPE_CLASS.TYPE_DATEANDTIME:
	
	convertResult := TryConvert_STRING_TO_DT(in, _DT);
	IF convertResult THEN
		convertAddress := ADR(_DT);
	END_IF
	
	__SYSTEM.TYPE_CLASS.TYPE_STRING:
	
	convertResult := TryConvert_STRING_TO_STRING(in, _STRING);
	IF convertResult THEN
		convertAddress := ADR(_STRING);
	END_IF
	
END_CASE

IF convertResult THEN
	memcpy(out.pValue,convertAddress,DINT_TO_UDINT(out.diSize));
END_IF

TryConvert_STRING_TO_Destination := convertResult;

END_FUNCTION

// ---- Converters/STRING_TO_/TryConvert_STRING_TO_WORD.TcPOU
FUNCTION TryConvert_STRING_TO_WORD : BOOL
VAR_INPUT
	in : STRING;
	out : REFERENCE TO WORD;
END_VAR

IF in <> WORD_TO_STRING(STRING_TO_WORD(in)) THEN
	RETURN;
END_IF

out := STRING_TO_WORD(in);
TryConvert_STRING_TO_WORD := TRUE;

END_FUNCTION

// ---- Converters/STRING_TO_/TryConvert_STRING_TO_DWORD.TcPOU
FUNCTION TryConvert_STRING_TO_DWORD : BOOL
VAR_INPUT
	in : STRING;
	out : REFERENCE TO DWORD;
END_VAR

IF in <> DWORD_TO_STRING(STRING_TO_DWORD(in)) THEN
	RETURN;
END_IF

out := STRING_TO_DWORD(in);
TryConvert_STRING_TO_DWORD := TRUE;

END_FUNCTION

// ---- Converters/STRING_TO_/TryConvert_STRING_TO_LWORD.TcPOU
FUNCTION TryConvert_STRING_TO_LWORD : BOOL
VAR_INPUT
	in : STRING;
	out : REFERENCE TO LWORD;
END_VAR

IF in <> LWORD_TO_STRING(STRING_TO_LWORD(in)) THEN
	RETURN;
END_IF

out := STRING_TO_LWORD(in);
TryConvert_STRING_TO_LWORD := TRUE;

END_FUNCTION

// ---- Converters/STRING_TO_/TryConvert_STRING_TO_SINT.TcPOU
FUNCTION TryConvert_STRING_TO_SINT : BOOL
VAR_INPUT
	in : STRING;
	out : REFERENCE TO SINT;
END_VAR

IF in <> SINT_TO_STRING(STRING_TO_SINT(in)) THEN
	RETURN;
END_IF

out := STRING_TO_SINT(in);
TryConvert_STRING_TO_SINT := TRUE;

END_FUNCTION

// ---- Converters/STRING_TO_/TryConvert_STRING_TO_INT.TcPOU
FUNCTION TryConvert_STRING_TO_INT : BOOL
VAR_INPUT
	in : STRING;
	out : REFERENCE TO INT;
END_VAR

IF in <> INT_TO_STRING(STRING_TO_INT(in)) THEN
	RETURN;
END_IF

out := STRING_TO_INT(in);
TryConvert_STRING_TO_INT := TRUE;

END_FUNCTION

// ---- Converters/STRING_TO_/TryConvert_STRING_TO_DINT.TcPOU
FUNCTION TryConvert_STRING_TO_DINT : BOOL
VAR_INPUT
	in : STRING;
	out : REFERENCE TO DINT;
END_VAR

IF in <> DINT_TO_STRING(STRING_TO_DINT(in)) THEN
	RETURN;
END_IF

out := STRING_TO_DINT(in);
TryConvert_STRING_TO_DINT := TRUE;

END_FUNCTION

// ---- Converters/STRING_TO_/TryConvert_STRING_TO_LINT.TcPOU
FUNCTION TryConvert_STRING_TO_LINT : BOOL
VAR_INPUT
	in : STRING;
	out : REFERENCE TO LINT;
END_VAR

IF in <> LINT_TO_STRING(STRING_TO_LINT(in)) THEN
	RETURN;
END_IF

out := STRING_TO_LINT(in);
TryConvert_STRING_TO_LINT := TRUE;

END_FUNCTION

// ---- Converters/STRING_TO_/TryConvert_STRING_TO_USINT.TcPOU
FUNCTION TryConvert_STRING_TO_USINT : BOOL
VAR_INPUT
	in : STRING;
	out : REFERENCE TO USINT;
END_VAR

IF in <> USINT_TO_STRING(STRING_TO_USINT(in)) THEN
	RETURN;
END_IF

out := STRING_TO_USINT(in);
TryConvert_STRING_TO_USINT := TRUE;

END_FUNCTION

// ---- Converters/STRING_TO_/TryConvert_STRING_TO_UINT.TcPOU
FUNCTION TryConvert_STRING_TO_UINT : BOOL
VAR_INPUT
	in : STRING;
	out : REFERENCE TO UINT;
END_VAR

IF in <> UINT_TO_STRING(STRING_TO_UINT(in)) THEN
	RETURN;
END_IF

out := STRING_TO_UINT(in);
TryConvert_STRING_TO_UINT := TRUE;

END_FUNCTION

// ---- Converters/STRING_TO_/TryConvert_STRING_TO_UDINT.TcPOU
FUNCTION TryConvert_STRING_TO_UDINT : BOOL
VAR_INPUT
	in : STRING;
	out : REFERENCE TO UDINT;
END_VAR

IF in <> UDINT_TO_STRING(STRING_TO_UDINT(in)) THEN
	RETURN;
END_IF

out := STRING_TO_UDINT(in);
TryConvert_STRING_TO_UDINT := TRUE;

END_FUNCTION

// ---- Converters/STRING_TO_/TryConvert_STRING_TO_ULINT.TcPOU
FUNCTION TryConvert_STRING_TO_ULINT : BOOL
VAR_INPUT
	in : STRING;
	out : REFERENCE TO ULINT;
END_VAR

IF in <> ULINT_TO_STRING(STRING_TO_ULINT(in)) THEN
	RETURN;
END_IF

out := STRING_TO_ULINT(in);
TryConvert_STRING_TO_ULINT := TRUE;

END_FUNCTION

// ---- Converters/STRING_TO_/TryConvert_STRING_TO_REAL.TcPOU
FUNCTION TryConvert_STRING_TO_REAL : BOOL
VAR_INPUT
	in : STRING;
	out : REFERENCE TO REAL;
END_VAR

IF in <> REAL_TO_STRING(STRING_TO_REAL(in)) THEN
	RETURN;
END_IF

out := STRING_TO_REAL(in);
TryConvert_STRING_TO_REAL := TRUE;

END_FUNCTION

// ---- Converters/STRING_TO_/TryConvert_STRING_TO_LREAL.TcPOU
FUNCTION TryConvert_STRING_TO_LREAL : BOOL
VAR_INPUT
	in : STRING;
	out : REFERENCE TO LREAL;
END_VAR

IF in <> LREAL_TO_STRING(STRING_TO_LREAL(in)) THEN
	RETURN;
END_IF

out := STRING_TO_LREAL(in);
TryConvert_STRING_TO_LREAL := TRUE;

END_FUNCTION

// ---- Converters/STRING_TO_/TryConvert_STRING_TO_TIME.TcPOU
FUNCTION TryConvert_STRING_TO_TIME : BOOL
VAR_INPUT
	in : STRING;
	out : REFERENCE TO TIME;
END_VAR

IF in <> TIME_TO_STRING(STRING_TO_TIME(in)) THEN
	RETURN;
END_IF

out := STRING_TO_TIME(in);
TryConvert_STRING_TO_TIME := TRUE;

END_FUNCTION

// ---- Converters/STRING_TO_/TryConvert_STRING_TO_TOD.TcPOU
FUNCTION TryConvert_STRING_TO_TOD : BOOL
VAR_INPUT
	in : STRING;
	out : REFERENCE TO TOD;
END_VAR

IF in <> TOD_TO_STRING(STRING_TO_TOD(in)) THEN
	RETURN;
END_IF

out := STRING_TO_TOD(in);
TryConvert_STRING_TO_TOD := TRUE;

END_FUNCTION

// ---- Converters/STRING_TO_/TryConvert_STRING_TO_DT.TcPOU
FUNCTION TryConvert_STRING_TO_DT : BOOL
VAR_INPUT
	in : STRING;
	out : REFERENCE TO DT;
END_VAR

IF in <> DT_TO_STRING(STRING_TO_DT(in)) THEN
	RETURN;
END_IF

out := STRING_TO_DT(in);
TryConvert_STRING_TO_DT := TRUE;

END_FUNCTION

// ---- Converters/STRING_TO_/TryConvert_STRING_TO_STRING.TcPOU
FUNCTION TryConvert_STRING_TO_STRING : BOOL
VAR_INPUT
	in : STRING;
	out : REFERENCE TO STRING;
END_VAR

out := in;
TryConvert_STRING_TO_STRING := TRUE;

END_FUNCTION

// ---- Converters/TIME_TO_/TryConvert_TIME_TO_BOOL.TcPOU
FUNCTION TryConvert_TIME_TO_BOOL : BOOL
VAR_INPUT
	in : TIME;
	out : REFERENCE TO BOOL;
END_VAR

out := TIME_TO_BOOL(in);
TryConvert_TIME_TO_BOOL := TRUE;

END_FUNCTION

// ---- Converters/TIME_TO_/TryConvert_TIME_TO_BYTE.TcPOU
FUNCTION TryConvert_TIME_TO_BYTE : BOOL
VAR_INPUT
	in : TIME;
	out : REFERENCE TO BYTE;
END_VAR

IF in > DatatypeLimits.MAX_VALUE_OF_TIME_WHICH_CAN_BE_HELD_IN_A_BYTE THEN
	RETURN;
END_IF

out := TIME_TO_BYTE(in);
TryConvert_TIME_TO_BYTE := TRUE;

END_FUNCTION

// ---- Converters/TIME_TO_/TryConvert_TIME_TO_DATE.TcPOU
FUNCTION TryConvert_TIME_TO_DATE : BOOL
VAR_INPUT
	in : TIME;
	out : REFERENCE TO DATE;
END_VAR

out := TIME_TO_DATE(in);
TryConvert_TIME_TO_DATE := TRUE;

END_FUNCTION

// ---- Converters/TIME_TO_/TryConvert_TIME_TO_Destination.TcPOU
FUNCTION TryConvert_TIME_TO_Destination : BOOL
VAR_INPUT
	in : TIME;
	out : ANY;
END_VAR
VAR
	convertResult : BOOL := FALSE;
	convertAddress : PVOID;
	_BOOL : BOOL;
	_BYTE : BYTE;
	_WORD : WORD;
	_DWORD : DWORD;
	_LWORD : LWORD;
	_SINT : SINT;
	_INT : INT;
	_DINT : DINT;
	_LINT : LINT;
	_USINT : USINT;
	_UINT : UINT;
	_UDINT : UDINT;
	_ULINT : ULINT;
	_REAL : REAL;
	_LREAL : LREAL;
	_TIME : TIME;
	_TOD : TOD;
	_DATE : DATE;
	_DT : DT;
	_STRING : STRING;
END_VAR

CASE out.TypeClass OF
	__SYSTEM.TYPE_CLASS.TYPE_BOOL:
	
	convertResult := TryConvert_TIME_TO_BOOL(in, _BOOL);
	IF convertResult THEN
		convertAddress := ADR(_BOOL);
	END_IF
	
	__SYSTEM.TYPE_CLASS.TYPE_BYTE:
	
	convertResult := TryConvert_TIME_TO_BYTE(in, _BYTE);
	IF convertResult THEN
		convertAddress := ADR(_BYTE);
	END_IF
	
	__SYSTEM.TYPE_CLASS.TYPE_WORD:
	
	convertResult := TryConvert_TIME_TO_WORD(in, _WORD);
	IF convertResult THEN
		convertAddress := ADR(_WORD);
	END_IF
	
	__SYSTEM.TYPE_CLASS.TYPE_DWORD:
	
	convertResult := TryConvert_TIME_TO_DWORD(in, _DWORD);
	IF convertResult THEN
		convertAddress := ADR(_DWORD);
	END_IF
	
	__SYSTEM.TYPE_CLASS.TYPE_LWORD:
	
	convertResult := TryConvert_TIME_TO_LWORD(in, _LWORD);
	IF convertResult THEN
		convertAddress := ADR(_LWORD);
	END_IF
	
	__SYSTEM.TYPE_CLASS.TYPE_SINT:
	
	convertResult := TryConvert_TIME_TO_SINT(in, _SINT);
	IF convertResult THEN
		convertAddress := ADR(_SINT);
	END_IF
	
	__SYSTEM.TYPE_CLASS.TYPE_INT:
	
	convertResult := TryConvert_TIME_TO_INT(in, _INT);
	IF convertResult THEN
		convertAddress := ADR(_INT);
	END_IF
	
	__SYSTEM.TYPE_CLASS.TYPE_DINT:
	
	convertResult := TryConvert_TIME_TO_DINT(in, _DINT);
	IF convertResult THEN
		convertAddress := ADR(_DINT);
	END_IF
	
	__SYSTEM.TYPE_CLASS.TYPE_LINT:
	
	convertResult := TryConvert_TIME_TO_LINT(in, _LINT);
	IF convertResult THEN
		convertAddress := ADR(_LINT);
	END_IF
	
	__SYSTEM.TYPE_CLASS.TYPE_USINT:
	
	convertResult := TryConvert_TIME_TO_USINT(in, _USINT);
	IF convertResult THEN
		convertAddress := ADR(_USINT);
	END_IF
	
	__SYSTEM.TYPE_CLASS.TYPE_UINT:
	
	convertResult := TryConvert_TIME_TO_UINT(in, _UINT);
	IF convertResult THEN
		convertAddress := ADR(_UINT);
	END_IF
	
	__SYSTEM.TYPE_CLASS.TYPE_UDINT:
	
	convertResult := TryConvert_TIME_TO_UDINT(in, _UDINT);
	IF convertResult THEN
		convertAddress := ADR(_UDINT);
	END_IF
	
	__SYSTEM.TYPE_CLASS.TYPE_ULINT:
	
	convertResult := TryConvert_TIME_TO_ULINT(in, _ULINT);
	IF convertResult THEN
		convertAddress := ADR(_ULINT);
	END_IF
	
	__SYSTEM.TYPE_CLASS.TYPE_REAL:
	
	convertResult := TryConvert_TIME_TO_REAL(in, _REAL);
	IF convertResult THEN
		convertAddress := ADR(_REAL);
	END_IF
	
	__SYSTEM.TYPE_CLASS.TYPE_LREAL:
	
	convertResult := TryConvert_TIME_TO_LREAL(in, _LREAL);
	IF convertResult THEN
		convertAddress := ADR(_LREAL);
	END_IF
	
	__SYSTEM.TYPE_CLASS.TYPE_TIME:
	
	convertResult := TryConvert_TIME_TO_TIME(in, _TIME);
	IF convertResult THEN
		convertAddress := ADR(_TIME);
	END_IF
	
	__SYSTEM.TYPE_CLASS.TYPE_TIMEOFDAY:
	
	convertResult := TryConvert_TIME_TO_TOD(in, _TOD);
	IF convertResult THEN
		convertAddress := ADR(_TOD);
	END_IF
	
	__SYSTEM.TYPE_CLASS.TYPE_DATE:
	
	convertResult := TryConvert_TIME_TO_DATE(in, _DATE);
	IF convertResult THEN
		convertAddress := ADR(_DATE);
	END_IF
	
	__SYSTEM.TYPE_CLASS.TYPE_DATEANDTIME:
	
	convertResult := TryConvert_TIME_TO_DT(in, _DT);
	IF convertResult THEN
		convertAddress := ADR(_DT);
	END_IF
	
	__SYSTEM.TYPE_CLASS.TYPE_STRING:
	
	convertResult := TryConvert_TIME_TO_STRING(in, _STRING);
	IF convertResult THEN
		convertAddress := ADR(_STRING);
	END_IF
	
END_CASE

IF convertResult THEN
	memcpy(out.pValue,convertAddress,DINT_TO_UDINT(out.diSize));
END_IF

TryConvert_TIME_TO_Destination := convertResult;

END_FUNCTION

// ---- Converters/TIME_TO_/TryConvert_TIME_TO_WORD.TcPOU
FUNCTION TryConvert_TIME_TO_WORD : BOOL
VAR_INPUT
	in : TIME;
	out : REFERENCE TO WORD;
END_VAR

IF in > DatatypeLimits.MAX_VALUE_OF_TIME_WHICH_CAN_BE_HELD_IN_A_WORD THEN
	RETURN;
END_IF

out := TIME_TO_WORD(in);
TryConvert_TIME_TO_WORD := TRUE;

END_FUNCTION

// ---- Converters/TIME_TO_/TryConvert_TIME_TO_DWORD.TcPOU
FUNCTION TryConvert_TIME_TO_DWORD : BOOL
VAR_INPUT
	in : TIME;
	out : REFERENCE TO DWORD;
END_VAR

out := TIME_TO_DWORD(in);
TryConvert_TIME_TO_DWORD := TRUE;

END_FUNCTION

// ---- Converters/TIME_TO_/TryConvert_TIME_TO_LWORD.TcPOU
FUNCTION TryConvert_TIME_TO_LWORD : BOOL
VAR_INPUT
	in : TIME;
	out : REFERENCE TO LWORD;
END_VAR

out := TIME_TO_LWORD(in);
TryConvert_TIME_TO_LWORD := TRUE;

END_FUNCTION

// ---- Converters/TIME_TO_/TryConvert_TIME_TO_SINT.TcPOU
FUNCTION TryConvert_TIME_TO_SINT : BOOL
VAR_INPUT
	in : TIME;
	out : REFERENCE TO SINT;
END_VAR

IF in > DatatypeLimits.MAX_VALUE_OF_TIME_WHICH_CAN_BE_HELD_IN_A_SINT THEN
	RETURN;
END_IF

out := TIME_TO_SINT(in);
TryConvert_TIME_TO_SINT := TRUE;

END_FUNCTION

// ---- Converters/TIME_TO_/TryConvert_TIME_TO_INT.TcPOU
FUNCTION TryConvert_TIME_TO_INT : BOOL
VAR_INPUT
	in : TIME;
	out : REFERENCE TO INT;
END_VAR

IF in > DatatypeLimits.MAX_VALUE_OF_TIME_WHICH_CAN_BE_HELD_IN_A_INT THEN
	RETURN;
END_IF

out := TIME_TO_INT(in);
TryConvert_TIME_TO_INT := TRUE;

END_FUNCTION

// ---- Converters/TIME_TO_/TryConvert_TIME_TO_DINT.TcPOU
FUNCTION TryConvert_TIME_TO_DINT : BOOL
VAR_INPUT
	in : TIME;
	out : REFERENCE TO DINT;
END_VAR

IF in > DatatypeLimits.MAX_VALUE_OF_TIME_WHICH_CAN_BE_HELD_IN_A_DINT THEN
	RETURN;
END_IF

out := TIME_TO_DINT(in);
TryConvert_TIME_TO_DINT := TRUE;

END_FUNCTION

// ---- Converters/TIME_TO_/TryConvert_TIME_TO_LINT.TcPOU
FUNCTION TryConvert_TIME_TO_LINT : BOOL
VAR_INPUT
	in : TIME;
	out : REFERENCE TO LINT;
END_VAR

out := TIME_TO_LINT(in);
TryConvert_TIME_TO_LINT := TRUE;

END_FUNCTION

// ---- Converters/TIME_TO_/TryConvert_TIME_TO_USINT.TcPOU
FUNCTION TryConvert_TIME_TO_USINT : BOOL
VAR_INPUT
	in : TIME;
	out : REFERENCE TO USINT;
END_VAR

IF in > DatatypeLimits.MAX_VALUE_OF_TIME_WHICH_CAN_BE_HELD_IN_A_USINT THEN
	RETURN;
END_IF

out := TIME_TO_USINT(in);
TryConvert_TIME_TO_USINT := TRUE;

END_FUNCTION

// ---- Converters/TIME_TO_/TryConvert_TIME_TO_UINT.TcPOU
FUNCTION TryConvert_TIME_TO_UINT : BOOL
VAR_INPUT
	in : TIME;
	out : REFERENCE TO UINT;
END_VAR

IF in > DatatypeLimits.MAX_VALUE_OF_TIME_WHICH_CAN_BE_HELD_IN_A_UINT THEN
	RETURN;
END_IF

out := TIME_TO_UINT(in);
TryConvert_TIME_TO_UINT := TRUE;

END_FUNCTION

// ---- Converters/TIME_TO_/TryConvert_TIME_TO_UDINT.TcPOU
FUNCTION TryConvert_TIME_TO_UDINT : BOOL
VAR_INPUT
	in : TIME;
	out : REFERENCE TO UDINT;
END_VAR

out := TIME_TO_UDINT(in);
TryConvert_TIME_TO_UDINT := TRUE;

END_FUNCTION

// ---- Converters/TIME_TO_/TryConvert_TIME_TO_ULINT.TcPOU
FUNCTION TryConvert_TIME_TO_ULINT : BOOL
VAR_INPUT
	in : TIME;
	out : REFERENCE TO ULINT;
END_VAR

out := TIME_TO_ULINT(in);
TryConvert_TIME_TO_ULINT := TRUE;

END_FUNCTION

// ---- Converters/TIME_TO_/TryConvert_TIME_TO_REAL.TcPOU
FUNCTION TryConvert_TIME_TO_REAL : BOOL
VAR_INPUT
	in : TIME;
	out : REFERENCE TO REAL;
END_VAR

out := TIME_TO_REAL(in);
TryConvert_TIME_TO_REAL := TRUE;

END_FUNCTION

// ---- Converters/TIME_TO_/TryConvert_TIME_TO_LREAL.TcPOU
FUNCTION TryConvert_TIME_TO_LREAL : BOOL
VAR_INPUT
	in : TIME;
	out : REFERENCE TO LREAL;
END_VAR

out := TIME_TO_LREAL(in);
TryConvert_TIME_TO_LREAL := TRUE;

END_FUNCTION

// ---- Converters/TIME_TO_/TryConvert_TIME_TO_TIME.TcPOU
FUNCTION TryConvert_TIME_TO_TIME : BOOL
VAR_INPUT
	in : TIME;
	out : REFERENCE TO TIME;
END_VAR

out := in;
TryConvert_TIME_TO_TIME := TRUE;

END_FUNCTION

// ---- Converters/TIME_TO_/TryConvert_TIME_TO_TOD.TcPOU
FUNCTION TryConvert_TIME_TO_TOD : BOOL
VAR_INPUT
	in : TIME;
	out : REFERENCE TO TOD;
END_VAR

IF in > DatatypeLimits.MAX_VALUE_OF_TIME_WHICH_CAN_BE_HELD_IN_A_TOD THEN
	RETURN;
END_IF

out := TIME_TO_TOD(in);
TryConvert_TIME_TO_TOD := TRUE;

END_FUNCTION

// ---- Converters/TIME_TO_/TryConvert_TIME_TO_DT.TcPOU
FUNCTION TryConvert_TIME_TO_DT : BOOL
VAR_INPUT
	in : TIME;
	out : REFERENCE TO DT;
END_VAR

out := TIME_TO_DT(in);
TryConvert_TIME_TO_DT := TRUE;

END_FUNCTION

// ---- Converters/TIME_TO_/TryConvert_TIME_TO_STRING.TcPOU
FUNCTION TryConvert_TIME_TO_STRING : BOOL
VAR_INPUT
	in : TIME;
	out : REFERENCE TO STRING;
END_VAR

out := TIME_TO_STRING(in);
TryConvert_TIME_TO_STRING := TRUE;

END_FUNCTION

// ---- Converters/TryConvert_Source_TO_Destination.TcPOU
{attribute 'linkalways'} 
FUNCTION TryConvert_Source_TO_Destination : BOOL
VAR_INPUT
	in : ANY;
	out : ANY;
END_VAR
VAR
	_BOOL : BOOL;
	_BYTE : BYTE;
	_WORD : WORD;
	_DWORD : DWORD;
	_LWORD : LWORD;
	_SINT : SINT;
	_INT : INT;
	_DINT : DINT;
	_LINT : LINT;
	_USINT : USINT;
	_UINT : UINT;
	_UDINT : UDINT;
	_ULINT : ULINT;
	_REAL : REAL;
	_LREAL : LREAL;
	_TIME : TIME;
	_TOD : TOD;
	_DATE : DATE;
	_DT : DT;
	_STRING : STRING;
	convertResult : BOOL := FALSE;
END_VAR

CASE in.TypeClass OF

	__SYSTEM.TYPE_CLASS.TYPE_BOOL :
		memcpy(ADR(_BOOL),in.pValue,DINT_TO_UDINT(in.diSize));
		convertResult := TryConvert_BOOL_To_Destination(_BOOL, out);
		
	__SYSTEM.TYPE_CLASS.TYPE_BYTE :
		memcpy(ADR(_BYTE),in.pValue,DINT_TO_UDINT(in.diSize));
		convertResult := TryConvert_BYTE_To_Destination(_BYTE, out);
		
	__SYSTEM.TYPE_CLASS.TYPE_WORD :
		memcpy(ADR(_WORD),in.pValue,DINT_TO_UDINT(in.diSize));
		convertResult := TryConvert_WORD_To_Destination(_WORD, out);
		
	__SYSTEM.TYPE_CLASS.TYPE_DWORD :
		memcpy(ADR(_DWORD),in.pValue,DINT_TO_UDINT(in.diSize));
		convertResult := TryConvert_DWORD_To_Destination(_DWORD, out);
		
	__SYSTEM.TYPE_CLASS.TYPE_LWORD :
		memcpy(ADR(_LWORD),in.pValue,DINT_TO_UDINT(in.diSize));
		convertResult := TryConvert_LWORD_To_Destination(_LWORD, out);
		
	__SYSTEM.TYPE_CLASS.TYPE_SINT :
		memcpy(ADR(_SINT),in.pValue,DINT_TO_UDINT(in.diSize));
		convertResult := TryConvert_SINT_To_Destination(_SINT, out);
		
	__SYSTEM.TYPE_CLASS.TYPE_INT :
		memcpy(ADR(_INT),in.pValue,DINT_TO_UDINT(in.diSize));
		convertResult := TryConvert_INT_To_Destination(_INT, out);
		
	__SYSTEM.TYPE_CLASS.TYPE_DINT :
		memcpy(ADR(_DINT),in.pValue,DINT_TO_UDINT(in.diSize));
		convertResult := TryConvert_DINT_To_Destination(_DINT, out);
		
	__SYSTEM.TYPE_CLASS.TYPE_LINT :
		memcpy(ADR(_LINT),in.pValue,DINT_TO_UDINT(in.diSize));
		convertResult := TryConvert_LINT_To_Destination(_LINT, out);
		
	__SYSTEM.TYPE_CLASS.TYPE_USINT :
		memcpy(ADR(_USINT),in.pValue,DINT_TO_UDINT(in.diSize));
		convertResult := TryConvert_USINT_To_Destination(_USINT, out);
		
	__SYSTEM.TYPE_CLASS.TYPE_UINT :
		memcpy(ADR(_UINT),in.pValue,DINT_TO_UDINT(in.diSize));
		convertResult := TryConvert_UINT_To_Destination(_UINT, out);
		
	__SYSTEM.TYPE_CLASS.TYPE_UDINT :
		memcpy(ADR(_UDINT),in.pValue,DINT_TO_UDINT(in.diSize));
		convertResult := TryConvert_UDINT_To_Destination(_UDINT, out);
		
	__SYSTEM.TYPE_CLASS.TYPE_ULINT :
		memcpy(ADR(_ULINT),in.pValue,DINT_TO_UDINT(in.diSize));
		convertResult := TryConvert_ULINT_To_Destination(_ULINT, out);
		
	__SYSTEM.TYPE_CLASS.TYPE_REAL :
		memcpy(ADR(_REAL),in.pValue,DINT_TO_UDINT(in.diSize));
		convertResult := TryConvert_REAL_To_Destination(_REAL, out);
		
	__SYSTEM.TYPE_CLASS.TYPE_LREAL :
		memcpy(ADR(_LREAL),in.pValue,DINT_TO_UDINT(in.diSize));
		convertResult := TryConvert_LREAL_To_Destination(_LREAL, out);
		
	__SYSTEM.TYPE_CLASS.TYPE_TIME :
		memcpy(ADR(_TIME),in.pValue,DINT_TO_UDINT(in.diSize));
		convertResult := TryConvert_TIME_To_Destination(_TIME, out);
		
	__SYSTEM.TYPE_CLASS.TYPE_TIMEOFDAY :
		memcpy(ADR(_TOD),in.pValue,DINT_TO_UDINT(in.diSize));
		convertResult := TryConvert_TOD_To_Destination(_TOD, out);
		
	__SYSTEM.TYPE_CLASS.TYPE_DATE :
		memcpy(ADR(_DATE),in.pValue,DINT_TO_UDINT(in.diSize));
		convertResult := TryConvert_DATE_To_Destination(_DATE, out);
		
	__SYSTEM.TYPE_CLASS.TYPE_DATEANDTIME :
		memcpy(ADR(_DT),in.pValue,DINT_TO_UDINT(in.diSize));
		convertResult := TryConvert_DT_To_Destination(_DT, out);
		
	__SYSTEM.TYPE_CLASS.TYPE_STRING :
		memcpy(ADR(_STRING),in.pValue,DINT_TO_UDINT(in.diSize));
		convertResult := TryConvert_STRING_To_Destination(_STRING, out);
		
	END_CASE
TryConvert_Source_TO_Destination  := convertResult;

END_FUNCTION
